(* IEC 61131-3 sources: ElnaAutomator/ExampleProject/FunctionBlocks, 19 files *)

(* ---- fb_AI_Init.st ---- *)
FUNCTION_BLOCK fb_AI_Init

VAR_INPUT
	data_Ini : BOOL; (*Флаг необходимости инициализации параметров.*)
	dLL : LREAL;
	dHL : LREAL;
	dLA : LREAL;
	dHA : LREAL;
	dLW : LREAL;
	dHW : LREAL;
	ISVALIDREF_LA : BOOL   := False;
	ISVALIDREF_HA : BOOL   := False;
	ISVALIDREF_LW : BOOL   := False;
	ISVALIDREF_HW : BOOL   := False;
	delayLA : TIME   := T#0S;
	delayLW : TIME   := T#0S;
	delayHW : TIME   := T#0S;
	delayHA : TIME   := T#0S;
	inpLL : LREAL   := 4000.0;
	inpHL : LREAL   := 20000.0;
	CurrentShotCircuit : LREAL   := 21000.0;
	CurrentBreakCircuit : LREAL   := 3700.0;
	maxChangeSpeed : LREAL;
	maxChangeSpeedDown : LREAL;
	histeresis : LREAL;
	aperturFilter : LREAL;
	exponentialFilter : LREAL;
	rassoglasovanie : LREAL;
	inOpcCommandsDisabled : BOOL;
END_VAR

VAR_IN_OUT
	strAI : struct_AI; (*Дескриптор AI-канала.*)
END_VAR

VAR_OUTPUT
	Init : BOOL   := FALSE; (*Флаг успешно выполненной инициализации.*)
END_VAR

(*****            Функциональный блок переинициализации структуры-дескриптора канала аналогового ввода.            *****)
     Init := false;

    IF data_Ini THEN                            (* Параметрам требуется переинициализация. *)
        strAI.dLL                := dLL;
        strAI.dHL                := dHL;
        strAI.dLA                := dLA;
        strAI.dHA                := dHA;
        strAI.dLW                := dLW;
        strAI.dHW                := dHW;
        strAI.ISVALIDREF_LA      := ISVALIDREF_LA;
        strAI.ISVALIDREF_HA      := ISVALIDREF_HA;
        strAI.ISVALIDREF_LW      := ISVALIDREF_LW;
        strAI.ISVALIDREF_HW      := ISVALIDREF_HW;
        strAI.delayLA            := delayLA;
        strAI.delayLW            := delayLW;
        strAI.delayHW            := delayHW;
        strAI.delayHA            := delayHA;
        strAI.inpLL              := inpLL;
        strAI.inpHL              := inpHL;
        strAI.CurrentShotCircuit := CurrentShotCircuit;
        strAI.CurrentBreakCircuit:= CurrentBreakCircuit;
        strAI.maxChangeSpeed     := maxChangeSpeed;
        strAI.maxChangeSpeedDown := maxChangeSpeedDown;
        strAI.histeresis         := histeresis;
        strAI.aperturFilter      := aperturFilter;
        strAI.exponentialFilter  := exponentialFilter;
        strAI.rassoglasovanie    := rassoglasovanie;
        strAI.rassoglasovanie    := rassoglasovanie;

        data_Ini:=false;
        Init := TRUE;
     END_IF;
  IF Init THEN
        dLL:= 0.0;
        dHL:= 0.0;
        dLA:= 0.0;
        dHA:= 0.0;
        dLW:= 0.0;
        dHW:= 0.0;
        inpLL:= 4000.0;
        inpHL:= 20000.0;
        CurrentShotCircuit:= 21000.0;
        CurrentBreakCircuit:= 3700.0;
        ISVALIDREF_LA:= false;
        ISVALIDREF_HA:= false;
        ISVALIDREF_LW:= false;
        ISVALIDREF_HW:= false;
        delayLA:= T#0S;
        delayLW:= T#0S;
        delayHW:= T#0S;
        delayHA:= T#0S;
        maxChangeSpeed:= 0.0;
        maxChangeSpeedDown:= 0.0;
        histeresis:= 0.0;
        aperturFilter:= 0.0;
        exponentialFilter:= 0.0;
        rassoglasovanie:= 0.0;
      END_IF;

(* ---- fb_AiSourceMlp.st ---- *)
FUNCTION_BLOCK fb_AiSourceMlp

VAR_INPUT
	arAIN : TItemAIN; (*Данные от модуля AI*)
	err_mod : TItemDIN; (*Диагностика от модуля AI*)
END_VAR

VAR_IN_OUT
	strAI : struct_AI; (*Текущие параметры канала AI*)
END_VAR

VAR
	_statusAi : TYPE_StatusAi;
	_commandAnalog : TYPE_CommandAnalog;
	_sunpackerCommand : fb_sunpackerCommand;
	_AnalogLimitFlags : TYPE_AnalogLimitFlags;
	notReliable : BOOL;
	_lastValue : LREAL;
	resetCmdTimer : TON;
	_LastValueTimer : TON;
	resetCmdTimerPriznak : BOOL;
	k : LREAL;
	b : LREAL;
	ap : LREAL;
	raznitsa : LREAL;
	rABS : LREAL;
	h : LREAL;
	mismatch : LREAL;
	parametr : BYTE;
	source : BYTE;
	cmd : BYTE;
	lastCmd : BYTE;
	source_for_Status : BYTE;
	cmd_for_Status : BYTE;
	command_error_for_Status : BYTE;
	onInit : BOOL;
	off_trig : R_TRIG;
	on_trig : R_TRIG;
	remont_trig : R_TRIG;
	LL_trig : R_TRIG;
	HL_trig : R_TRIG;
	Normal_trig : R_TRIG;
	Nedostover_trig : R_TRIG;
END_VAR

strAI.opcCommandsDisabled := strAI.inopcCommandsDisabled ;

(* ---- При первом пуске принимаем значение уставок ---- *)
IF NOT onInit THEN

          strAI.LL := strAI.dLL;
          strAI.HL := strAI.dHL;

          IF strAI.ISVALIDREF_HA THEN strAI.HA := strAI.dHA; END_IF;

          IF strAI.ISVALIDREF_LA THEN strAI.LA := strAI.dLA; END_IF;

          IF strAI.ISVALIDREF_HW THEN strAI.HW := strAI.dHW; END_IF;

          IF strAI.ISVALIDREF_LW THEN strAI.LW := strAI.dLW; END_IF;

	onInit  := TRUE;
END_IF;

(* ---- пересчет тока в физ величину ---- *)
k := (strAI.HL - strAI.LL)/(strAI.inpHl - strAI.inpLL);
b := strAI.LL - k * strAI.inpLL;
strAI.value := k * arAIN.dblValue + b;

(* ---- определение обрыва и кз ----- *)

strAI.blConnect :=(*(UINT_TO_WORD(arAIN.wFlags) = 1472) and*) (UINT_TO_WORD(err_mod.wValue) = 20) and (UINT_TO_WORD(err_mod.wFlags) = 192);
IF NOT strAI.blConnect THEN
    strAI.interval := _statusAi.NOTDEFINED;
ELSIF ((arAIN.dblValue < strAI.currentBreakCircuit) AND (strAI.currentBreakCircuit > 0.0)) OR ((strAI.interval = _statusAi.LL) AND (arAIN.dblValue < (strAI.currentBreakCircuit + 100.0))) THEN
    strAI.interval := _statusAi.LL;
ELSIF ((arAIN.dblValue > strAI.currentShotCircuit) AND (strAI.currentShotCircuit > 0.0)) OR ((strAI.interval = _statusAi.HL) AND (arAIN.dblValue > (strAI.currentShotCircuit - 100.0))) THEN
    strAI.interval := _statusAi.HL;
ELSE
    strAI.interval := _statusAi.normal;
END_IF;

IF NOT strAI.imit THEN
	(* Расчет апертурного фильтра*)
	ap := strAI.aperturFilter * 0.01 * (strAI.HL - strAI.LL);
	IF strAI.aperturFilter <> 0.0 THEN raznitsa := strAI.value- _lastValue;
		IF 	raznitsa < 0.0 	THEN 	rABS := -raznitsa; 		ELSE 	rABS := raznitsa; 		END_IF;
		IF 	rABS > ap 	THEN 	strAI.value := strAI.value;	ELSE 	strAI.value := _lastValue; 	END_IF;
	END_IF;

	(* Расчет экпоненциального фильтра*)
	IF strAI.exponentialFilter <> 0.0 THEN strAI.value := (strAI.exponentialFilter * strAI.value) + ((1.0 - strAI.exponentialFilter) * _lastValue); END_IF;
ELSE
	strAI.interval := _statusAi.normal;
END_IF;

IF notReliable THEN strAI.interval := _statusAi.NOTRELIABLE; END_IF;

IF NOT notReliable THEN
	IF strAI.interval >= _statusAi.normal THEN
		strAI.interval := _statusAi.NOTDEFINED;
		h := strAI.histeresis* 0.01 * (strAI.HL-strAI.LL);
		(*определение выхода за аппаратные границы вынесено в GetData.здесь только для нужд имитации*)
		IF strAI.imit THEN
			mismatch := strAI.rassoglasovanie * 0.01 * (strAI.HL - strAI.LL);
			IF ( strAI.value < strAI.LL - mismatch)   THEN strAI.interval := _statusAi.LL;
			ELSIF  (strAI.value > strAI.Hl + mismatch) THEN strAI.interval := _statusAi.HL; END_IF;
		ELSE
			strAI.interval := _statusAi.normal;
			IF strAI.ISVALIDREF_LA AND NOT strAI.Disabled_LA AND (strAI.interval = _statusAi.normal) THEN
				IF (strAI.value  < strAI.LA) OR ((strAI.interval = _statusAi.LA)  AND ((strAI.value - h) < strAI.LA))  THEN
					strAI.interval := _statusAi.LA;
				END_IF;
			END_IF;
			IF strAI.ISVALIDREF_HA  AND NOT strAI.Disabled_HA AND (strAI.interval = _statusAi.normal)  THEN
				IF (strAI.value > strAI.HA) OR ((strAI.interval = _statusAi.HA)  AND ((strAI.value + h) > strAI.HA))  THEN
					strAI.interval := _statusAi.HA;
				END_IF;
			END_IF;
			IF strAI.ISVALIDREF_LW AND NOT strAI.Disabled_LW AND (strAI.interval = _statusAi.normal)  THEN
				IF (strAI.value < strAI.LW) OR ((strAI.interval = _statusAi.LW)  AND ((strAI.value - h) < strAI.LW)) THEN
					strAI.interval := _statusAi.LW;
				END_IF;
			END_IF;
			IF strAI.ISVALIDREF_HW AND NOT strAI.Disabled_HW  AND (strAI.interval = _statusAi.normal) THEN
				IF (strAI.value > strAI.HW)  OR ((strAI.interval = _statusAi.HW)  AND ((strAI.value + h) > strAI.HW))   THEN
					strAI.interval := _statusAi.HW;
				END_IF;
			END_IF;
		END_IF;
	END_IF;
ELSE
	strAI.interval := _statusAi.NOTRELIABLE;
END_IF;

IF strAI.remont THEN strAI.interval := _statusAi.NOTDEFINED; END_IF;

(* ---- Если управление с ВУ заблокировано, то  передаем команду из алгоритма ---- *)
IF strAI.inOpcCommandsDisabled THEN
	strAI.inCommand := strAI.inCommand_Alg;
ELSE (* иначе передаем команду с АРМа*)
	strAI.inCommand := strAI.inCommand_ARM;
END_IF;

_sunpackerCommand(command := strAI.inCommand);
	source := _sunpackerCommand.source;
	parametr := _sunpackerCommand.parametr;
	cmd := _sunpackerCommand.cmd;

IF cmd <> 0 AND lastCmd <> cmd and (((NOT strAI.opcCommandsDisabled) AND source > 0) OR source = 0) then
	CASE BYTE_TO_INT(cmd) OF
	(*cmd_SetUstavki*) 1 :
				IF ((parametr AND _AnalogLimitFlags.LL) <> 0)		             	THEN 	strAI.LL := strAI.dLL; END_IF;
				IF ((parametr AND _AnalogLimitFlags.HL) <> 0)		 	          THEN	strAI.HL := strAI.dHL; END_IF;
				IF ((parametr AND _AnalogLimitFlags.LA) <> 0) AND strAI.ISVALIDREF_LA 	THEN	strAI.LA := strAI.dLA; END_IF;
				IF ((parametr AND _AnalogLimitFlags.HA) <> 0) AND strAI.ISVALIDREF_HA 	THEN	strAI.HA := strAI.dHA; END_IF;
				IF ((parametr AND _AnalogLimitFlags.LW) <> 0) AND strAI.ISVALIDREF_LW 	THEN	strAI.LW := strAI.dLW; END_IF;
				IF ((parametr AND _AnalogLimitFlags.HW) <> 0) AND strAI.ISVALIDREF_HW 	THEN	strAI.HW := strAI.dHW; END_IF;
	(*cmd_SetRemont*) 6 :
				strAI.remont := TRUE;
	(*cmd_ResetRemont*) 7 :
				strAI.remont := FALSE;
	(*cmd_kvitNotReliable*) 4 :
				notReliable := FALSE;
	END_CASE;
	source_for_Status := source;
	cmd_for_Status := cmd;
	command_error_for_Status := 0;
	resetCmdTimer(IN := FALSE);
	resetCmdTimerPriznak := TRUE;
END_IF;
lastCmd := cmd;

resetCmdTimer(IN := resetCmdTimerPriznak, PT := T#5S);
IF resetCmdTimer.Q THEN
	resetCmdTimerPriznak := FALSE;
	source_for_Status := 0;
	cmd_for_Status := 0;
	command_error_for_Status := 0;
END_IF;

strAI.NS_Min := (strAI.value < strAI.minValue) AND strAI.minValue_ISVALIDREF;
strAI.NS_Max := (strAI.value > strAI.maxValue) AND strAI.maxValue_ISVALIDREF;

strAI.NS := (strAI.interval <= _statusAi.normal) AND NOT strAI.remont;

Normal_trig(CLK := strAI.interval >= _statusAi.normal);

IF NOT Normal_trig.Q THEN
	_LastValueTimer(PT := T#1S);
	IF (strAI.value<>_lastValue) OR _LastValueTimer.Q THEN
		IF (_LastValueTimer.ET>T#0MS) THEN
			strAI.ChangeSpeed:=(strAI.value-_lastValue)/(TIME_TO_LREAL(_LastValueTimer.ET));
		END_IF;
		_LastValueTimer(IN:=FALSE);

		_LastValueTimer(IN:=TRUE);
	END_IF;
END_IF;
_lastValue := strAI.value;

IF ((strAI.maxChangeSpeed<>0.0) OR  (strAI.maxChangeSpeedDown<>0.0)) AND ( strAI.interval>=_statusAi.normal) THEN
		IF (strAI.ChangeSpeed>0.0) THEN
		    IF (strAI.ChangeSpeed > strAI.maxChangeSpeed) AND (strAI.maxChangeSpeed>0.0000001) THEN
			 notReliable:=TRUE;
		    END_IF;
		ELSE
		    IF (ABS(strAI.ChangeSpeed)>strAI.maxChangeSpeedDown) AND (strAI.maxChangeSpeedDown>0.0000001)  THEN
                               notReliable:=TRUE;
		    END_IF;
		END_IF;

END_IF;

strAI.status := SHL(BYTE_TO_DWORD(source_for_Status), 29) 		              (* Источник команды *)
			OR SHL(BYTE_TO_DWORD(cmd_for_Status), 26) 	    (* Команда *)
			OR SHL(BYTE_TO_DWORD(command_error_for_Status), 23)   (* Ошибка команды *)
			OR SHL(BOOL_TO_DWORD(strAI.OpcCommandsDisabled ), 21) (* Управление в ВУ заблокировано *)
			OR SHL(BOOL_TO_DWORD(strAI.Disabled_HA), 9)		    (* ВА исключена из формирования интервала *)
			OR SHL(BOOL_TO_DWORD(strAI.Disabled_LA), 8)		    (* НА исключена из формирования интервала *)
			OR SHL(BOOL_TO_DWORD(strAI.Disabled_HW), 7)		    (* ВП исключена из формирования интервала *)
			OR SHL(BOOL_TO_DWORD(strAI.Disabled_LW), 6)	              (* НП исключена из формирования интервала *)
			OR SHL(BOOL_TO_DWORD(strAI.NS), 5)			    (* неиспарвность сигнала *)
			OR SHL(BOOL_TO_DWORD(strAI.remont), 4)	              (* Выведен в ремонт *)
			OR BYTE_TO_DWORD(strAI.interval);	              (* интервал *)

(* ---- Opc_Ai_get.st ---- *)
FUNCTION_BLOCK Opc_Ai_get

VAR_EXTERNAL
	Ai : AiConfig;
	AI_A1_newHW : LREAL;
	AI_A1_newHA : LREAL;
	AI_A1_newLA : LREAL;
	AI_A1_newLW : LREAL;
	AI_A1_newHL : LREAL;
	AI_A1_newLL : LREAL;
	AI_A1_command : UINT;
	AI_A2_newHW : LREAL;
	AI_A2_newHA : LREAL;
	AI_A2_newLA : LREAL;
	AI_A2_newLW : LREAL;
	AI_A2_newHL : LREAL;
	AI_A2_newLL : LREAL;
	AI_A2_command : UINT;
END_VAR

Ai.A1.dHW := AI_A1_newHW;
Ai.A1.dHA := AI_A1_newHA;
Ai.A1.dLA := AI_A1_newLA;
Ai.A1.dLW := AI_A1_newLW;
Ai.A1.dHL := AI_A1_newHL;
Ai.A1.dLL := AI_A1_newLL;
Ai.A1.inCommand_ARM := UINT_TO_WORD(AI_A1_command);

Ai.A2.dHW := AI_A2_newHW;
Ai.A2.dHA := AI_A2_newHA;
Ai.A2.dLA := AI_A2_newLA;
Ai.A2.dLW := AI_A2_newLW;
Ai.A2.dHL := AI_A2_newHL;
Ai.A2.dLL := AI_A2_newLL;
Ai.A2.inCommand_ARM := UINT_TO_WORD(AI_A2_command);

(* ---- Opc_Ai_init.st ---- *)
FUNCTION_BLOCK Opc_Ai_init

VAR_EXTERNAL
	Ai : AiConfig;
	AI_A1_HW : LREAL;
	AI_A1_newHW : LREAL;
	AI_A1_HA : LREAL;
	AI_A1_newHA : LREAL;
	AI_A1_LA : LREAL;
	AI_A1_newLA : LREAL;
	AI_A1_LW : LREAL;
	AI_A1_newLW : LREAL;
	AI_A1_HL : LREAL;
	AI_A1_newHL : LREAL;
	AI_A1_LL : LREAL;
	AI_A1_newLL : LREAL;
	AI_A2_HW : LREAL;
	AI_A2_newHW : LREAL;
	AI_A2_HA : LREAL;
	AI_A2_newHA : LREAL;
	AI_A2_LA : LREAL;
	AI_A2_newLA : LREAL;
	AI_A2_LW : LREAL;
	AI_A2_newLW : LREAL;
	AI_A2_HL : LREAL;
	AI_A2_newHL : LREAL;
	AI_A2_LL : LREAL;
	AI_A2_newLL : LREAL;
END_VAR

AI_A1_HW := Ai.A1.HW;
AI_A1_newHW := Ai.A1.dHW;
AI_A1_HA := Ai.A1.HA;
AI_A1_newHA := Ai.A1.dHA;
AI_A1_LA := Ai.A1.LA;
AI_A1_newLA := Ai.A1.dLA;
AI_A1_LW := Ai.A1.LW;
AI_A1_newLW := Ai.A1.dLW;
AI_A1_LL := Ai.A1.LL;
AI_A1_newLL := Ai.A1.dLL;
AI_A1_HL := Ai.A1.HL;
AI_A1_newHL := Ai.A1.dHL;

AI_A2_HW := Ai.A2.HW;
AI_A2_newHW := Ai.A2.dHW;
AI_A2_HA := Ai.A2.HA;
AI_A2_newHA := Ai.A2.dHA;
AI_A2_LA := Ai.A2.LA;
AI_A2_newLA := Ai.A2.dLA;
AI_A2_LW := Ai.A2.LW;
AI_A2_newLW := Ai.A2.dLW;
AI_A2_LL := Ai.A2.LL;
AI_A2_newLL := Ai.A2.dLL;
AI_A2_HL := Ai.A2.HL;
AI_A2_newHL := Ai.A2.dHL;

(* ---- Opc_Ai_set.st ---- *)
FUNCTION_BLOCK Opc_Ai_set

VAR_EXTERNAL
	Ai : AiConfig;
	AI_A1_HW : LREAL;
	AI_A1_HA : LREAL;
	AI_A1_LA : LREAL;
	AI_A1_LW : LREAL;
	AI_A1_HL : LREAL;
	AI_A1_LL : LREAL;
	AI_A1_value : LREAL;
	AI_A1_status : UDINT;
	AI_A2_HW : LREAL;
	AI_A2_HA : LREAL;
	AI_A2_LA : LREAL;
	AI_A2_LW : LREAL;
	AI_A2_HL : LREAL;
	AI_A2_LL : LREAL;
	AI_A2_value : LREAL;
	AI_A2_status : UDINT;
END_VAR

AI_A1_HW := Ai.A1.HW;
AI_A1_HA := Ai.A1.HA;
AI_A1_LA := Ai.A1.LA;
AI_A1_LW := Ai.A1.LW;
AI_A1_LL := Ai.A1.LL;
AI_A1_HL := Ai.A1.HL;
AI_A1_value := Ai.A1.value;
AI_A1_status := DWORD_TO_UDINT(Ai.A1.status);

AI_A2_HW := Ai.A2.HW;
AI_A2_HA := Ai.A2.HA;
AI_A2_LA := Ai.A2.LA;
AI_A2_LW := Ai.A2.LW;
AI_A2_LL := Ai.A2.LL;
AI_A2_HL := Ai.A2.HL;
AI_A2_value := Ai.A2.value;
AI_A2_status := DWORD_TO_UDINT(Ai.A2.status);

(* ---- Opc_Im_get.st ---- *)
FUNCTION_BLOCK Opc_Im_get

VAR_EXTERNAL
	Im : ImConfig;
	Im_Kran1_inCommand_ARM : UINT;
	Im_Kran4_inCommand_ARM : UINT;
	Im_Kran2_inCommand_ARM : UINT;
	Im_Kran3_inCommand_ARM : UINT;
	Im_Nu_inCommand_ARM : UINT;
	Im_Nu2_inCommand_ARM : UINT;
	Im_Avom1_inCommand_ARM : UINT;
	Im_Avom2_inCommand_ARM : UINT;
	Im_Avom3_inCommand_ARM : UINT;
	Im_Avom4_inCommand_ARM : UINT;
	Im_Mv_inCommand_ARM : UINT;
	Im_SectionSwitch1_inCommand_ARM : UINT;
END_VAR

Im.Kran1.inCommand_ARM := UINT_TO_WORD(Im_Kran1_inCommand_ARM);

Im.Kran4.inCommand_ARM := UINT_TO_WORD(Im_Kran4_inCommand_ARM);

Im.Kran2.inCommand_ARM := UINT_TO_WORD(Im_Kran2_inCommand_ARM);

Im.Kran3.inCommand_ARM := UINT_TO_WORD(Im_Kran3_inCommand_ARM);

Im.Nu.inCommand_ARM := UINT_TO_WORD(Im_Nu_inCommand_ARM);

Im.Nu2.inCommand_ARM := UINT_TO_WORD(Im_Nu2_inCommand_ARM);

Im.Avom1.inCommand_ARM := UINT_TO_WORD(Im_Avom1_inCommand_ARM);

Im.Avom2.inCommand_ARM := UINT_TO_WORD(Im_Avom2_inCommand_ARM);

Im.Avom3.inCommand_ARM := UINT_TO_WORD(Im_Avom3_inCommand_ARM);

Im.Avom4.inCommand_ARM := UINT_TO_WORD(Im_Avom4_inCommand_ARM);

Im.Mv.inCommand_ARM := UINT_TO_WORD(Im_Mv_inCommand_ARM);

Im.SectionSwitch1.inCommand_ARM := UINT_TO_WORD(Im_SectionSwitch1_inCommand_ARM);

(* ---- Opc_Im_set.st ---- *)
FUNCTION_BLOCK Opc_Im_set

VAR_EXTERNAL
	Im : ImConfig;
	Im_Kran1_status : UDINT;
	Im_Kran4_status : UDINT;
	Im_Kran2_status : UDINT;
	Im_Kran3_status : UDINT;
	Im_Nu_status : UDINT;
	Im_Nu2_status : UDINT;
	Im_Avom1_status : UDINT;
	Im_Avom2_status : UDINT;
	Im_Avom3_status : UDINT;
	Im_Avom4_status : UDINT;
	Im_Mv_status : UDINT;
	Im_SectionSwitch1_status : UDINT;
	Im_SingleSignals_SI0_status : UDINT;
	Im_SingleSignals_SI1_status : UDINT;
	Im_SingleSignals_SI2_status : UDINT;
	Im_SingleSignals_SI3_status : UDINT;
	Im_SingleSignals_SI4_status : UDINT;
	Im_SingleSignals_SI5_status : UDINT;
	Im_SingleSignals_SI6_status : UDINT;
END_VAR

Im_Kran1_status := DWORD_TO_UDINT(Im.Kran1.status);

Im_Kran4_status := DWORD_TO_UDINT(Im.Kran4.status);

Im_Kran2_status := DWORD_TO_UDINT(Im.Kran2.status);

Im_Kran3_status := DWORD_TO_UDINT(Im.Kran3.status);

Im_Nu_status := DWORD_TO_UDINT(Im.Nu.status);

Im_Nu2_status := DWORD_TO_UDINT(Im.Nu2.status);

Im_Avom1_status := DWORD_TO_UDINT(Im.Avom1.status);

Im_Avom2_status := DWORD_TO_UDINT(Im.Avom2.status);

Im_Avom3_status := DWORD_TO_UDINT(Im.Avom3.status);

Im_Avom4_status := DWORD_TO_UDINT(Im.Avom4.status);

Im_Mv_status := DWORD_TO_UDINT(Im.Mv.status);

Im_SectionSwitch1_status := DWORD_TO_UDINT(Im.SectionSwitch1.status);

Im_SingleSignals_SI0_status := DWORD_TO_UDINT(Im.SingleSignals.SI0.status);

Im_SingleSignals_SI1_status := DWORD_TO_UDINT(Im.SingleSignals.SI1.status);

Im_SingleSignals_SI2_status := DWORD_TO_UDINT(Im.SingleSignals.SI2.status);

Im_SingleSignals_SI3_status := DWORD_TO_UDINT(Im.SingleSignals.SI3.status);

Im_SingleSignals_SI4_status := DWORD_TO_UDINT(Im.SingleSignals.SI4.status);

Im_SingleSignals_SI5_status := DWORD_TO_UDINT(Im.SingleSignals.SI5.status);

Im_SingleSignals_SI6_status := DWORD_TO_UDINT(Im.SingleSignals.SI6.status);

(* ---- Opc_Protections_get.st ---- *)
FUNCTION_BLOCK Opc_Protections_get

VAR_EXTERNAL
	Protections : ProtectionsConfig;
	Protections_Ap1_inCommand_ARM : UINT;
	Protections_AiP1_inCommand_ARM : UINT;
	Protections_AiP2_inCommand_ARM : UINT;
	Protections_AiP3_inCommand_ARM : UINT;
	Protections_DiP1_inCommand_ARM : UINT;
	Protections_DiP2_inCommand_ARM : UINT;
	Protections_DiP3_inCommand_ARM : UINT;
	Protections_DiP4_inCommand_ARM : UINT;
	Protections_DiP5_inCommand_ARM : UINT;
END_VAR

Protections.Ap1.inCommand_ARM := UINT_TO_WORD(Protections_Ap1_inCommand_ARM);

Protections.AiP1.inCommand_ARM := UINT_TO_WORD(Protections_AiP1_inCommand_ARM);

Protections.AiP2.inCommand_ARM := UINT_TO_WORD(Protections_AiP2_inCommand_ARM);

Protections.AiP3.inCommand_ARM := UINT_TO_WORD(Protections_AiP3_inCommand_ARM);

Protections.DiP1.inCommand_ARM := UINT_TO_WORD(Protections_DiP1_inCommand_ARM);

Protections.DiP2.inCommand_ARM := UINT_TO_WORD(Protections_DiP2_inCommand_ARM);

Protections.DiP3.inCommand_ARM := UINT_TO_WORD(Protections_DiP3_inCommand_ARM);

Protections.DiP4.inCommand_ARM := UINT_TO_WORD(Protections_DiP4_inCommand_ARM);

Protections.DiP5.inCommand_ARM := UINT_TO_WORD(Protections_DiP5_inCommand_ARM);

(* ---- Opc_Protections_set.st ---- *)
FUNCTION_BLOCK Opc_Protections_set

VAR_EXTERNAL
	Protections : ProtectionsConfig;
	Protections_Ap1_status : UDINT;
	Protections_AiP1_status : UDINT;
	Protections_AiP2_status : UDINT;
	Protections_AiP3_status : UDINT;
	Protections_DiP1_status : UDINT;
	Protections_DiP2_status : UDINT;
	Protections_DiP3_status : UDINT;
	Protections_DiP4_status : UDINT;
	Protections_DiP5_status : UDINT;
END_VAR

Protections_Ap1_status := DWORD_TO_UDINT(Protections.Ap1.status);

Protections_AiP1_status := DWORD_TO_UDINT(Protections.AiP1.status);

Protections_AiP2_status := DWORD_TO_UDINT(Protections.AiP2.status);

Protections_AiP3_status := DWORD_TO_UDINT(Protections.AiP3.status);

Protections_DiP1_status := DWORD_TO_UDINT(Protections.DiP1.status);

Protections_DiP2_status := DWORD_TO_UDINT(Protections.DiP2.status);

Protections_DiP3_status := DWORD_TO_UDINT(Protections.DiP3.status);

Protections_DiP4_status := DWORD_TO_UDINT(Protections.DiP4.status);

Protections_DiP5_status := DWORD_TO_UDINT(Protections.DiP5.status);

(* ---- Proc_Ai.st ---- *)
FUNCTION_BLOCK Proc_Ai

VAR
	fb_A1 : fb_AiSourceMlp;
	fb_A2 : fb_AiSourceMlp;
END_VAR

VAR_EXTERNAL
	Ai : AiConfig;
	arAIN_0 : TItemAIN;
	arAIN_1 : TItemAIN;
	AI_0_dblValue : LREAL;
	AI_1_dblValue : LREAL;
	arERR_0 : TItemDIN;;
END_VAR

fb_A1(arAIN := arAIN_0, strAI := Ai.A1, err_mod := arERR_0);
AI_0_dblValue := arAIN_0.dblValue;

fb_A2(arAIN := arAIN_1, strAI := Ai.A2, err_mod := arERR_0);
AI_1_dblValue := arAIN_1.dblValue;

(* ---- Proc_Ai_Init.st ---- *)
FUNCTION_BLOCK Proc_Ai_Init

VAR_INPUT
	init : BOOL;
END_VAR

VAR
	stAI_Ini : fb_AI_Init;
	inits : UINT;
END_VAR

VAR_INPUT
	initiales : UINT;
END_VAR

VAR_EXTERNAL
	Ai : AiConfig;
END_VAR

inits := 0;

stAI_Ini(data_Ini := TRUE, dLL := 0.0, dHL := 100.0,
ISVALIDREF_LW := TRUE, dLW := 20.0,
ISVALIDREF_HW := TRUE, dHW := 80.0,
ISVALIDREF_LA := TRUE, dLA := 10.0,
ISVALIDREF_HA := TRUE, dHA := 90.0,
strAI := Ai.A1);
inits := inits + BOOL_TO_UINT(stAI_Ini.Init);

stAI_Ini(data_Ini := TRUE, dLL := 0.0, dHL := 100.0,
ISVALIDREF_LW := TRUE, dLW := 20.0,
ISVALIDREF_HW := TRUE, dHW := 80.0,
ISVALIDREF_LA := TRUE, dLA := 10.0,
ISVALIDREF_HA := TRUE, dHA := 90.0,
strAI := Ai.A2);
inits := inits + BOOL_TO_UINT(stAI_Ini.Init);

initiales := 0;
IF init THEN initiales := inits; END_IF;

(* ---- Proc_Di.st ---- *)
FUNCTION_BLOCK Proc_Di

VAR
	fb_Di : fb_DiSourceMlp;
	fb_Di1 : fb_DiSourceMlp;
	fb_Di2 : fb_DiSourceMlp;
	fb_Di3 : fb_DiSourceMlp;
	fb_Di4 : fb_DiSourceMlp;
END_VAR

VAR_EXTERNAL
	di : DiConfig;
	arDIN_0 : TItemDIN;
	arDIN_1 : TItemDIN;
	arDIN_2 : TItemDIN;
	arDIN_3 : TItemDIN;
	arDIN_4 : TItemDIN;
	DI_0_1_wValue : UDINT;
	DI_2_3_wValue : UDINT;
	arERR_1 : TItemDIN;;
	arERR_2 : TItemDIN;;
	arERR_3 : TItemDIN;;
	arERR_4 : TItemDIN;;
	arERR_5 : TItemDIN;;
END_VAR

fb_Di(arDIN := arDIN_0, strDI := di.Di, err_mod := arERR_1);
fb_Di1(arDIN := arDIN_1, strDI := di.Di1, err_mod := arERR_2);
DI_0_1_wValue := DIwValue_Diag(arDIN_0.wValue, arDIN_1.wValue);

fb_Di2(arDIN := arDIN_2, strDI := di.Di2, err_mod := arERR_3);
fb_Di3(arDIN := arDIN_3, strDI := di.Di3, err_mod := arERR_4);
DI_2_3_wValue := DIwValue_Diag(arDIN_2.wValue, arDIN_3.wValue);

fb_Di4(arDIN := arDIN_4, strDI := di.Di4, err_mod := arERR_5);

(* ---- Proc_Di_Init.st ---- *)
FUNCTION_BLOCK Proc_Di_Init

VAR_INPUT
	init : BOOL;
END_VAR

VAR
	stDI_Ini : fb_DI_Init;
	inits : UINT;
END_VAR

VAR_INPUT
	initiales : UINT;
END_VAR

VAR_EXTERNAL
	di : DiConfig;
END_VAR

inits := 0;

stDI_Ini(data_Ini := TRUE, imit := FALSE, strDI := di.Di);
inits := inits + BOOL_TO_UINT(stDI_Ini.Init);

stDI_Ini(data_Ini := TRUE, imit := FALSE, strDI := di.Di1);
inits := inits + BOOL_TO_UINT(stDI_Ini.Init);

stDI_Ini(data_Ini := TRUE, imit := FALSE, strDI := di.Di2);
inits := inits + BOOL_TO_UINT(stDI_Ini.Init);

stDI_Ini(data_Ini := TRUE, imit := FALSE, strDI := di.Di3);
inits := inits + BOOL_TO_UINT(stDI_Ini.Init);

stDI_Ini(data_Ini := TRUE, imit := FALSE, strDI := di.Di4);
inits := inits + BOOL_TO_UINT(stDI_Ini.Init);

initiales := 0;
IF init THEN initiales := inits; END_IF;

(* ---- Proc_Do.st ---- *)
FUNCTION_BLOCK Proc_Do

VAR
	fb_Do1 : fb_DOSourceMlp;
	fb_Do2 : fb_DOSourceMlp;
	fb_Do3 : fb_DOSourceMlp;
	fb_Do4 : fb_DOSourceMlp;
	fb_Do5 : fb_DOSourceMlp;
END_VAR

VAR_EXTERNAL
	od : DoConfig;
	arDOUT_0 : TWordData;
	arDOUT_1 : TWordData;
	arDOUT_2 : TWordData;
	arDOUT_3 : TWordData;
	arDOUT_4 : TWordData;
	DO_0_wValue : UINT;
	DO_1_wValue : UINT;
	DO_2_wValue : UINT;
	DO_3_wValue : UINT;
	DO_4_wValue : UINT;
	arERR_1 : TItemDIN;;
	arERR_2 : TItemDIN;;
	arERR_3 : TItemDIN;;
	arERR_4 : TItemDIN;;
	arERR_5 : TItemDIN;;
END_VAR

fb_Do1(arDout := arDOUT_0, strDO := od.Do1, err_mod := arERR_1);
DO_0_wValue := arDOUT_0.wValue;

fb_Do2(arDout := arDOUT_1, strDO := od.Do2, err_mod := arERR_2);
DO_1_wValue := arDOUT_1.wValue;

fb_Do3(arDout := arDOUT_2, strDO := od.Do3, err_mod := arERR_3);
DO_2_wValue := arDOUT_2.wValue;

fb_Do4(arDout := arDOUT_3, strDO := od.Do4, err_mod := arERR_4);
DO_3_wValue := arDOUT_3.wValue;

fb_Do5(arDout := arDOUT_4, strDO := od.Do5, err_mod := arERR_5);
DO_4_wValue := arDOUT_4.wValue;

(*gpio_out not initialized*)

(* ---- Proc_Do_Init.st ---- *)
FUNCTION_BLOCK Proc_Do_Init

VAR_INPUT
	init : BOOL;
END_VAR

VAR
	stDO_Ini : fb_DO_Init;
	inits : UINT;
END_VAR

VAR_INPUT
	initiales : UINT;
END_VAR

VAR_EXTERNAL
	od : DoConfig;
END_VAR

inits := 0;

stDO_Ini(data_Ini := TRUE, imit := FALSE, strDO := od.Do1);
inits := inits + BOOL_TO_UINT(stDO_Ini.Init);

stDO_Ini(data_Ini := TRUE, imit := FALSE, strDO := od.Do2);
inits := inits + BOOL_TO_UINT(stDO_Ini.Init);

stDO_Ini(data_Ini := TRUE, imit := FALSE, strDO := od.Do3);
inits := inits + BOOL_TO_UINT(stDO_Ini.Init);

stDO_Ini(data_Ini := TRUE, imit := FALSE, strDO := od.Do4);
inits := inits + BOOL_TO_UINT(stDO_Ini.Init);

stDO_Ini(data_Ini := TRUE, imit := FALSE, strDO := od.Do5);
inits := inits + BOOL_TO_UINT(stDO_Ini.Init);

initiales := 0;
IF init THEN initiales := inits; END_IF;

(* ---- Proc_Im.st ---- *)
FUNCTION_BLOCK Proc_Im

VAR
	fb_Kran1 : fb_Kran;
	fb_Kran4 : fb_Kran;
	fb_Kran2 : fb_Kran;
	fb_Kran3 : fb_Kran;
	fb_Nu : fb_OilPump;
	fb_Nu2 : fb_OilPump;
	fb_Mv : fb_SectionSwitch;
	fb_SectionSwitch1 : fb_SectionSwitch;
	fb_Avom1 : fb_Switch;
	fb_Avom2 : fb_Switch;
	fb_Avom3 : fb_Switch;
	fb_Avom4 : fb_Switch;
	fb_So0 : fb_singleOutput;
	fb_So1 : fb_singleOutput;
	fb_So2 : fb_singleOutput;
	fb_So3 : fb_singleOutput;
	fb_So4 : fb_singleOutput;
	fb_So5 : fb_singleOutput;
	fb_So6 : fb_singleOutput;
	fb_So7 : fb_singleOutput;
	fb_SI0 : fb_singleSignal;
	fb_SI1 : fb_singleSignal;
	fb_SI2 : fb_singleSignal;
	fb_SI3 : fb_singleSignal;
	fb_SI4 : fb_singleSignal;
	fb_SI5 : fb_singleSignal;
	fb_SI6 : fb_singleSignal;
END_VAR

VAR_EXTERNAL
	di : DiConfig;
	od : DoConfig;
	Im : ImConfig;
END_VAR

fb_Kran1(statOn := di.Di.bits[1]._inversed,
statOn_reliability := di.Di.bits[1].reliability,
statOff := di.Di.bits[2]._inversed,
statOff_reliability := di.Di.bits[2].reliability,
cmdOn := od.Do1.bits[1],
cmdOff := od.Do2.bits[0],
inDp := di.Di1.bits[1],
inSo := di.Di.bits[3],
inSz := di.Di.bits[2],
strKr := Im.Kran1);

fb_Kran4(statOn := di.Di1.bits[2]._inversed,
statOn_reliability := di.Di1.bits[2].reliability,
statOff := di.Di2.bits[2]._inversed,
statOff_reliability := di.Di2.bits[2].reliability,
cmdOn := od.Do3.bits[2],
cmdOff := od.Do1.bits[2],
inDp := di.Di.bits[2],
inSo := di.Di2.bits[3],
inSz := di.Di1.bits[1],
strKr := Im.Kran4);

fb_Kran2(statOn := di.Di2.bits[3].value,
statOn_reliability := di.Di2.bits[3].reliability,
statOff := di.Di3.bits[1].value,
statOff_reliability := di.Di3.bits[1].reliability,
cmdOn := od.Do3.bits[3],
cmdOff := od.Do2.bits[3],
inDp := di.Di4.bits[3],
inSo := di.Di1.bits[1],
inSz := di.Di1.bits[2],
strKr := Im.Kran2);

fb_Kran3(statOn := di.Di3.bits[4]._inversed,
statOn_reliability := di.Di3.bits[4].reliability,
statOff := di.Di4.bits[3]._inversed,
statOff_reliability := di.Di4.bits[3].reliability,
cmdOn := od.Do2.bits[4],
cmdOff := od.Do3.bits[4],
inDp := di.Di4.bits[4],
inSo := di.Di1.bits[2],
inSz := di.Di4.bits[3],
strKr := Im.Kran3);

fb_Nu(statOn := di.Di.bits[1]._inversed,
statOn_reliability := di.Di.bits[1].reliability,
statOff := di.Di.bits[2]._inversed,
statOff_reliability := di.Di.bits[2].reliability,
cmdOn := od.Do2.bits[1],
cmdOff := od.Do1.bits[0],
inBreakCmdOn := di.Di.bits[3],
inBreakCmdOff := di.Di1.bits[4],
StrSw := Im.Nu);

fb_Nu2(statOn := di.Di2.bits[2].value,
statOn_reliability := di.Di2.bits[2].reliability,
statOff := di.Di3.bits[3].value,
statOff_reliability := di.Di3.bits[3].reliability,
cmdOn := od.Do4.bits[3],
cmdOff := od.Do1.bits[4],
inBreakCmdOn := di.Di.bits[4],
inBreakCmdOff := di.Di1.bits[3],
StrSw := Im.Nu2);

fb_Avom1(statOn := di.Di.bits[1].value,
statOn_reliability := di.Di.bits[1].reliability,
statOff := di.Di1.bits[2].value,
statOff_reliability := di.Di1.bits[2].reliability,
cmdOn := od.Do1.bits[1],
cmdOff := od.Do1.bits[0],
inBreakCmdOn := di.Di1.bits[2],
inBreakCmdOff := di.Di.bits[2],
StrSw := Im.Avom1);

fb_Avom2(statOn := di.Di3.bits[2]._inversed,
statOn_reliability := di.Di3.bits[2].reliability,
statOff := di.Di.bits[2]._inversed,
statOff_reliability := di.Di.bits[2].reliability,
cmdOn := od.Do4.bits[3],
cmdOff := od.Do2.bits[1],
inBreakCmdOn := di.Di1.bits[3],
inBreakCmdOff := di.Di1.bits[3],
StrSw := Im.Avom2);

fb_Avom3(statOn := di.Di1.bits[3]._inversed,
statOn_reliability := di.Di1.bits[3].reliability,
statOff := di.Di2.bits[3]._inversed,
statOff_reliability := di.Di2.bits[3].reliability,
cmdOn := od.Do1.bits[5],
cmdOff := od.Do3.bits[3],
inBreakCmdOn := di.Di3.bits[4],
inBreakCmdOff := di.Di2.bits[4],
StrSw := Im.Avom3);

fb_Avom4(statOn := di.Di.bits[4]._inversed,
statOn_reliability := di.Di.bits[4].reliability,
statOff := di.Di.bits[4]._inversed,
statOff_reliability := di.Di.bits[4].reliability,
cmdOn := od.Do2.bits[4],
cmdOff := od.Do3.bits[4],
inBreakCmdOn := di.Di3.bits[5],
inBreakCmdOff := di.Di4.bits[5],
StrSw := Im.Avom4);

fb_Mv(statOn := di.Di.bits[1]._inversed,
statOn_reliability := di.Di.bits[1].reliability,
statOff := di.Di.bits[2]._inversed,
statOff_reliability := di.Di.bits[2].reliability,
cmdOn := od.Do2.bits[1],
cmdOff := od.Do2.bits[0],
inBreakCmdOn := di.Di3.bits[4],
inBreakCmdOff := di.Di4.bits[3],
basketRolledin := di.Di.bits[2],
basketRolledout := di.Di.bits[3],
basketTest := di.Di1.bits[3],
StrSw := Im.Mv);

fb_SectionSwitch1(StrSw := Im.SectionSwitch1);

fb_SI0(signal := di.Di1.bits[1], str_SS := Im.SingleSignals.SI0);

fb_SI1(signal := di.Di1.bits[2], str_SS := Im.SingleSignals.SI1);

fb_SI2(signal := di.Di.bits[3], str_SS := Im.SingleSignals.SI2);

fb_SI3(signal := di.Di1.bits[4], str_SS := Im.SingleSignals.SI3);

fb_SI4(signal := di.Di3.bits[5], str_SS := Im.SingleSignals.SI4);

fb_SI5(signal := di.Di3.bits[6], str_SS := Im.SingleSignals.SI5);

fb_SI6(signal := di.Di4.bits[7], str_SS := Im.SingleSignals.SI6);

fb_So0(signal := od.Do1.bits[1], str_SO := Im.SingleOutputs.So0);

fb_So1(signal := od.Do2.bits[2], str_SO := Im.SingleOutputs.So1);

fb_So2(signal := od.Do3.bits[3], str_SO := Im.SingleOutputs.So2);

fb_So3(signal := od.Do1.bits[4], str_SO := Im.SingleOutputs.So3);

fb_So4(signal := od.Do2.bits[5], str_SO := Im.SingleOutputs.So4);

fb_So5(signal := od.Do1.bits[6], str_SO := Im.SingleOutputs.So5);

fb_So6(signal := od.Do1.bits[7], str_SO := Im.SingleOutputs.So6);

fb_So7(signal := od.Do2.bits[8], str_SO := Im.SingleOutputs.So7);

(* ---- Proc_Im_Init.st ---- *)
FUNCTION_BLOCK Proc_Im_Init

VAR_INPUT
	init : BOOL;
END_VAR

VAR
	stKr_Ini : fb_Kran_Init;
	stSw_Ini : fb_Switch_Init;
	stOp_Ini : fb_OilPump_Init;
	stSSw_Ini : fb_SectionSwitch_Init;
	stSs_Ini : fb_singleSignal_Init;
	stSo_Ini : fb_singleOutput_Init;
	inits : UINT;
END_VAR

VAR_INPUT
	initiales : UINT;
END_VAR

VAR_EXTERNAL
	Im : ImConfig;
END_VAR

stKr_Ini(str_Kr := Im.Kran1,
ISVALIDREF_inDp := TRUE,
ISVALIDREF_inSo := TRUE,
ISVALIDREF_inSz := TRUE,
ISVALIDREF_statOn := TRUE,
ISVALIDREF_statOff := TRUE,
ISVALIDREF_cmdOn := TRUE,
ISVALIDREF_cmdOff := TRUE);
inits := inits + BOOL_TO_UINT(stKr_Ini.Init);

stKr_Ini(str_Kr := Im.Kran4,
ISVALIDREF_inDp := TRUE,
ISVALIDREF_inSo := TRUE,
ISVALIDREF_inSz := TRUE,
ISVALIDREF_statOn := TRUE,
ISVALIDREF_statOff := TRUE,
ISVALIDREF_cmdOn := TRUE,
ISVALIDREF_cmdOff := TRUE);
inits := inits + BOOL_TO_UINT(stKr_Ini.Init);

stKr_Ini(str_Kr := Im.Kran2,
ISVALIDREF_inDp := TRUE,
ISVALIDREF_inSo := TRUE,
ISVALIDREF_inSz := TRUE,
ISVALIDREF_statOn := TRUE,
ISVALIDREF_statOff := TRUE,
ISVALIDREF_cmdOn := TRUE,
ISVALIDREF_cmdOff := TRUE);
inits := inits + BOOL_TO_UINT(stKr_Ini.Init);

stKr_Ini(str_Kr := Im.Kran3,
ISVALIDREF_inDp := TRUE,
ISVALIDREF_inSo := TRUE,
ISVALIDREF_inSz := TRUE,
ISVALIDREF_statOn := TRUE,
ISVALIDREF_statOff := TRUE,
ISVALIDREF_cmdOn := TRUE,
ISVALIDREF_cmdOff := TRUE);
inits := inits + BOOL_TO_UINT(stKr_Ini.Init);

stOp_Ini(str_Op := Im.Nu,
ISVALIDREF_inBreakCmdOn := TRUE,
ISVALIDREF_inBreakCmdOff := TRUE,
ISVALIDREF_statOn := TRUE,
ISVALIDREF_statOff := TRUE,
ISVALIDREF_cmdOn := TRUE,
ISVALIDREF_cmdOff := TRUE);
inits := inits + BOOL_TO_UINT(stOp_Ini.Init);

stOp_Ini(str_Op := Im.Nu2,
ISVALIDREF_inBreakCmdOn := TRUE,
ISVALIDREF_inBreakCmdOff := TRUE,
ISVALIDREF_statOn := TRUE,
ISVALIDREF_statOff := TRUE,
ISVALIDREF_cmdOn := TRUE,
ISVALIDREF_cmdOff := TRUE);
inits := inits + BOOL_TO_UINT(stOp_Ini.Init);

stSSw_Ini(str_Sw := Im.Mv,
ISVALIDREF_inBreakCmdOn := TRUE,
ISVALIDREF_inBreakCmdOff := TRUE,
ISVALIDREF_basketRolledIn := TRUE,
ISVALIDREF_basketRolledout := TRUE,
ISVALIDREF_basketTest := TRUE,
ISVALIDREF_statOn := TRUE,
ISVALIDREF_statOff := TRUE,
ISVALIDREF_cmdOn := TRUE,
ISVALIDREF_cmdOff := TRUE);
inits := inits + BOOL_TO_UINT(stSSw_Ini.Init);

stSSw_Ini(str_Sw := Im.SectionSwitch1);
inits := inits + BOOL_TO_UINT(stSSw_Ini.Init);

stSw_Ini(str_Sw := Im.Avom1,
ISVALIDREF_inBreakCmdOn := TRUE,
ISVALIDREF_inBreakCmdOff := TRUE,
ISVALIDREF_statOn := TRUE,
ISVALIDREF_statOff := TRUE,
ISVALIDREF_cmdOn := TRUE,
ISVALIDREF_cmdOff := TRUE);
inits := inits + BOOL_TO_UINT(stSw_Ini.Init);

stSw_Ini(str_Sw := Im.Avom2,
ISVALIDREF_inBreakCmdOn := TRUE,
ISVALIDREF_inBreakCmdOff := TRUE,
ISVALIDREF_statOn := TRUE,
ISVALIDREF_statOff := TRUE,
ISVALIDREF_cmdOn := TRUE,
ISVALIDREF_cmdOff := TRUE);
inits := inits + BOOL_TO_UINT(stSw_Ini.Init);

stSw_Ini(str_Sw := Im.Avom3,
ISVALIDREF_inBreakCmdOn := TRUE,
ISVALIDREF_inBreakCmdOff := TRUE,
ISVALIDREF_statOn := TRUE,
ISVALIDREF_statOff := TRUE,
ISVALIDREF_cmdOn := TRUE,
ISVALIDREF_cmdOff := TRUE);
inits := inits + BOOL_TO_UINT(stSw_Ini.Init);

stSw_Ini(str_Sw := Im.Avom4,
ISVALIDREF_inBreakCmdOn := TRUE,
ISVALIDREF_inBreakCmdOff := TRUE,
ISVALIDREF_statOn := TRUE,
ISVALIDREF_statOff := TRUE,
ISVALIDREF_cmdOn := TRUE,
ISVALIDREF_cmdOff := TRUE);
inits := inits + BOOL_TO_UINT(stSw_Ini.Init);

stSs_Ini(data_Ini := TRUE, inverse := FALSE, str_SS := Im.SingleSignals.SI0);
inits := inits + BOOL_TO_UINT(stSs_Ini.Init);

stSs_Ini(data_Ini := TRUE, inverse := FALSE, str_SS := Im.SingleSignals.SI1);
inits := inits + BOOL_TO_UINT(stSs_Ini.Init);

stSs_Ini(data_Ini := TRUE, inverse := FALSE, str_SS := Im.SingleSignals.SI2);
inits := inits + BOOL_TO_UINT(stSs_Ini.Init);

stSs_Ini(data_Ini := TRUE, inverse := FALSE, str_SS := Im.SingleSignals.SI3);
inits := inits + BOOL_TO_UINT(stSs_Ini.Init);

stSs_Ini(data_Ini := TRUE, inverse := FALSE, str_SS := Im.SingleSignals.SI4);
inits := inits + BOOL_TO_UINT(stSs_Ini.Init);

stSs_Ini(data_Ini := TRUE, inverse := FALSE, str_SS := Im.SingleSignals.SI5);
inits := inits + BOOL_TO_UINT(stSs_Ini.Init);

stSs_Ini(data_Ini := TRUE, inverse := FALSE, str_SS := Im.SingleSignals.SI6);
inits := inits + BOOL_TO_UINT(stSs_Ini.Init);

stSo_Ini(data_Ini := TRUE, inOpcCommandsDisabled := FALSE, str_SO := Im.SingleOutputs.So0);
inits := inits + BOOL_TO_UINT(stSo_Ini.Init);

stSo_Ini(data_Ini := TRUE, inOpcCommandsDisabled := FALSE, str_SO := Im.SingleOutputs.So1);
inits := inits + BOOL_TO_UINT(stSo_Ini.Init);

stSo_Ini(data_Ini := TRUE, inOpcCommandsDisabled := FALSE, str_SO := Im.SingleOutputs.So2);
inits := inits + BOOL_TO_UINT(stSo_Ini.Init);

stSo_Ini(data_Ini := TRUE, inOpcCommandsDisabled := FALSE, str_SO := Im.SingleOutputs.So3);
inits := inits + BOOL_TO_UINT(stSo_Ini.Init);

stSo_Ini(data_Ini := TRUE, inOpcCommandsDisabled := FALSE, str_SO := Im.SingleOutputs.So4);
inits := inits + BOOL_TO_UINT(stSo_Ini.Init);

stSo_Ini(data_Ini := TRUE, inOpcCommandsDisabled := FALSE, str_SO := Im.SingleOutputs.So5);
inits := inits + BOOL_TO_UINT(stSo_Ini.Init);

stSo_Ini(data_Ini := TRUE, inOpcCommandsDisabled := FALSE, str_SO := Im.SingleOutputs.So6);
inits := inits + BOOL_TO_UINT(stSo_Ini.Init);

stSo_Ini(data_Ini := TRUE, inOpcCommandsDisabled := FALSE, str_SO := Im.SingleOutputs.So7);
inits := inits + BOOL_TO_UINT(stSo_Ini.Init);

initiales := 0;
IF init THEN initiales := inits; END_IF;

(* ---- Proc_Protection.st ---- *)
FUNCTION_BLOCK Proc_Protection

VAR_EXTERNAL
	Protections : ProtectionsConfig;
	Ai : AiConfig;
	Im : ImConfig;
END_VAR

VAR
	fb_Ap1 : fb_AiProtection;
	fb_AiP1 : fb_AiProtection;
	fb_AiP2 : fb_AiProtection;
	fb_AiP3 : fb_AiProtection;
	fb_DiP1 : fb_DiProtection;
	fb_DiP2 : fb_DiProtection;
	fb_DiP3 : fb_DiProtection;
	fb_DiP4 : fb_DiProtection;
	fb_DiP5 : fb_DiProtection;
END_VAR

fb_Ap1(ai := Ai.A1, StrAIp := Protections.Ap1);

fb_AiP1(ai := Ai.A2, StrAIp := Protections.AiP1);

fb_AiP2(ai := Ai.A1, StrAIp := Protections.AiP2);

fb_AiP3(ai := Ai.A2, StrAIp := Protections.AiP3);

fb_DiP1(di := Im.SingleSignals.SI2, StrDIp := Protections.DiP1);

fb_DiP2(di := Im.SingleSignals.SI0, StrDIp := Protections.DiP2);

fb_DiP3(di := Im.SingleSignals.SI0, StrDIp := Protections.DiP3);

fb_DiP4(di := Im.SingleSignals.SI2, StrDIp := Protections.DiP4);

fb_DiP5(di := Im.SingleSignals.SI4, StrDIp := Protections.DiP5);

(* ---- Proc_Protections_Init.st ---- *)
FUNCTION_BLOCK Proc_Protections_Init

VAR_INPUT
	init : BOOL;
END_VAR

VAR
	stDIp_Ini : fb_DiProtection_Init;
	stAIp_Ini : fb_AiProtection_Init;
	inits : UINT;
END_VAR

VAR_INPUT
	initiales : UINT;
END_VAR

VAR_EXTERNAL
	Protections : ProtectionsConfig;
END_VAR

VAR
	_ProtectionTags : TYPE_ProtectionTags;
	_StatusAi : TYPE_StatusAi;
END_VAR

inits := 0;

stAIp_Ini(data_Ini := TRUE, delay := T#1S, inTag := _ProtectionTags.AOS, inRunOnStart := TRUE,
controlLimit := _StatusAi.LA, str_AIp := Protections.Ap1);
inits := inits + BOOL_TO_UINT(stAIp_Ini.Init);

stAIp_Ini(data_Ini := TRUE, delay := T#2S, inTag := _ProtectionTags.AOS, inRunOnStart := FALSE,
controlLimit := _StatusAi.HA, str_AIp := Protections.AiP1);
inits := inits + BOOL_TO_UINT(stAIp_Ini.Init);

stAIp_Ini(data_Ini := TRUE, delay := T#3S, inTag := _ProtectionTags.AOS, inRunOnStart := TRUE,
controlLimit := _StatusAi.LA, str_AIp := Protections.AiP2);
inits := inits + BOOL_TO_UINT(stAIp_Ini.Init);

stAIp_Ini(data_Ini := TRUE, delay := T#4S, inTag := _ProtectionTags.AOS, inRunOnStart := FALSE,
controlLimit := _StatusAi.HA, str_AIp := Protections.AiP3);
inits := inits + BOOL_TO_UINT(stAIp_Ini.Init);

stDIp_Ini(data_Ini := TRUE, delay := T#1S, inTag := _ProtectionTags.AOS, inRunOnStart := TRUE, str_DIp := Protections.DiP1);
inits := inits + BOOL_TO_UINT(stDIp_Ini.Init);

stDIp_Ini(data_Ini := TRUE, delay := T#2S, inTag := _ProtectionTags.AOS, inRunOnStart := TRUE, str_DIp := Protections.DiP2);
inits := inits + BOOL_TO_UINT(stDIp_Ini.Init);

stDIp_Ini(data_Ini := TRUE, delay := T#3S, inTag := _ProtectionTags.AOS, inRunOnStart := TRUE, str_DIp := Protections.DiP3);
inits := inits + BOOL_TO_UINT(stDIp_Ini.Init);

stDIp_Ini(data_Ini := TRUE, delay := T#4S, inTag := _ProtectionTags.AOS, inRunOnStart := FALSE, str_DIp := Protections.DiP4);
inits := inits + BOOL_TO_UINT(stDIp_Ini.Init);

stDIp_Ini(data_Ini := TRUE, delay := T#5S, inTag := _ProtectionTags.AOS, inRunOnStart := FALSE, str_DIp := Protections.DiP5);
inits := inits + BOOL_TO_UINT(stDIp_Ini.Init);

IF init THEN initiales := inits; END_IF;
